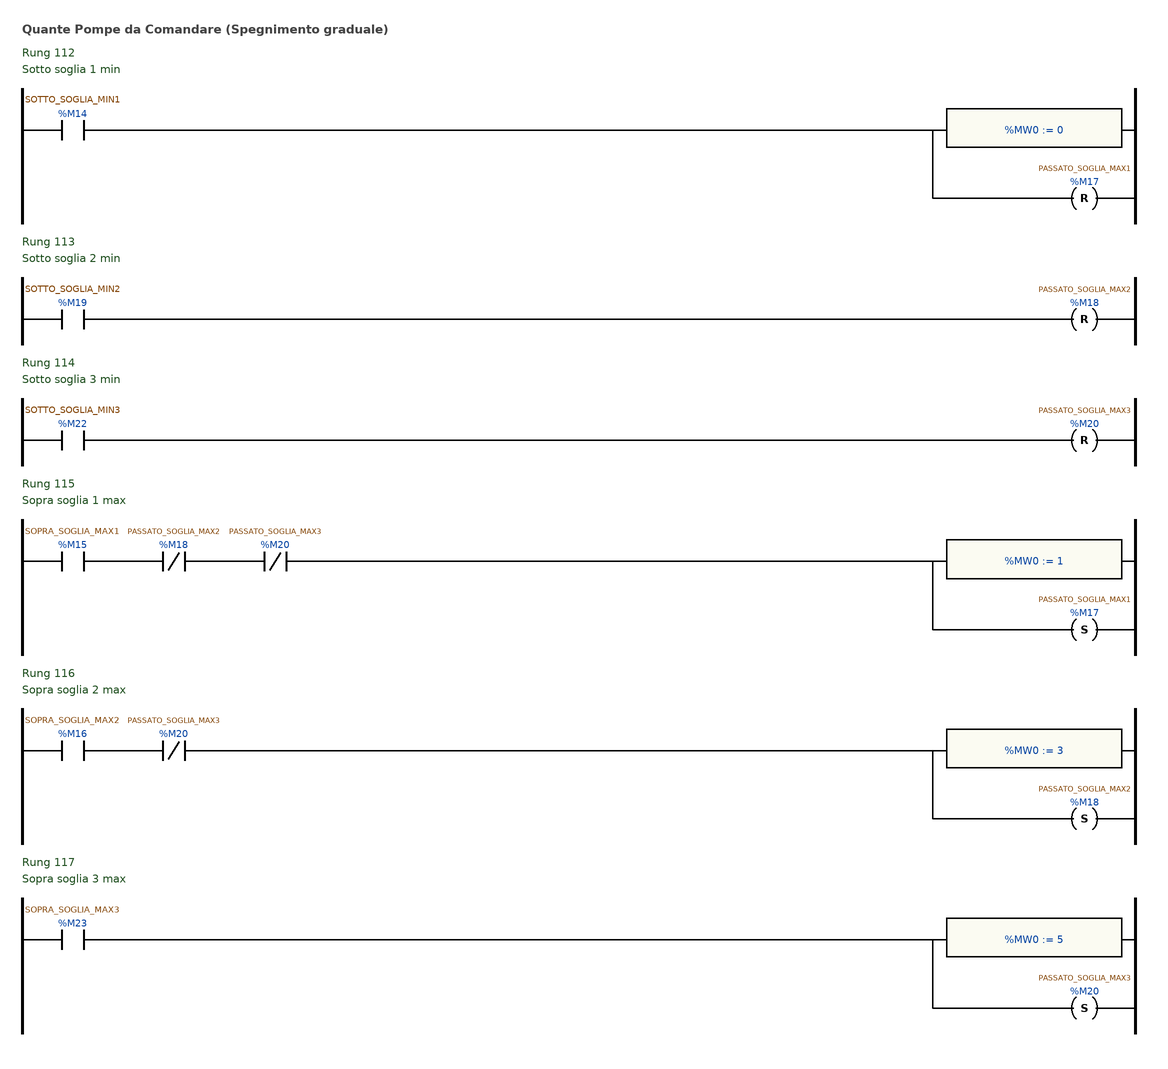
[picture p24: Quante Pompe da Comandare (Spegnimento graduale), ladder]

// Rung 112
// Sotto soglia 1 min
  LD %M14                 (* SOTTO_SOGLIA_MIN1 *)
  [ %MW0 := 0 ]           (* NUM_POMPE_DA_COMANDARE *)
  R %M17                  (* PASSATO_SOGLIA_MAX1 *)
  // as ST:
  //   IF SOTTO_SOGLIA_MIN1 THEN NUM_POMPE_DA_COMANDARE := 0; END_IF;
  //   IF SOTTO_SOGLIA_MIN1 THEN PASSATO_SOGLIA_MAX1 := FALSE; END_IF;

// Rung 113
// Sotto soglia 2 min
  LD %M19                 (* SOTTO_SOGLIA_MIN2 *)
  R %M18                  (* PASSATO_SOGLIA_MAX2 *)
  // as ST:
  //   IF SOTTO_SOGLIA_MIN2 THEN PASSATO_SOGLIA_MAX2 := FALSE; END_IF;

// Rung 114
// Sotto soglia 3 min
  LD %M22                 (* SOTTO_SOGLIA_MIN3 *)
  R %M20                  (* PASSATO_SOGLIA_MAX3 *)
  // as ST:
  //   IF SOTTO_SOGLIA_MIN3 THEN PASSATO_SOGLIA_MAX3 := FALSE; END_IF;

// Rung 115
// Sopra soglia 1 max
  LD %M15                 (* SOPRA_SOGLIA_MAX1 *)
  ANDN %M18               (* PASSATO_SOGLIA_MAX2 *)
  ANDN %M20               (* PASSATO_SOGLIA_MAX3 *)
  [ %MW0 := 1 ]           (* NUM_POMPE_DA_COMANDARE *)
  S %M17                  (* PASSATO_SOGLIA_MAX1 *)
  // as ST:
  //   IF SOPRA_SOGLIA_MAX1 AND NOT PASSATO_SOGLIA_MAX2 AND NOT PASSATO_SOGLIA_MAX3 THEN NUM_POMPE_DA_COMANDARE := 1; END_IF;
  //   IF SOPRA_SOGLIA_MAX1 AND NOT PASSATO_SOGLIA_MAX2 AND NOT PASSATO_SOGLIA_MAX3 THEN PASSATO_SOGLIA_MAX1 := TRUE; END_IF;

// Rung 116
// Sopra soglia 2 max
  LD %M16                 (* SOPRA_SOGLIA_MAX2 *)
  ANDN %M20               (* PASSATO_SOGLIA_MAX3 *)
  [ %MW0 := 3 ]           (* NUM_POMPE_DA_COMANDARE *)
  S %M18                  (* PASSATO_SOGLIA_MAX2 *)
  // as ST:
  //   IF SOPRA_SOGLIA_MAX2 AND NOT PASSATO_SOGLIA_MAX3 THEN NUM_POMPE_DA_COMANDARE := 3; END_IF;
  //   IF SOPRA_SOGLIA_MAX2 AND NOT PASSATO_SOGLIA_MAX3 THEN PASSATO_SOGLIA_MAX2 := TRUE; END_IF;

// Rung 117
// Sopra soglia 3 max
  LD %M23                 (* SOPRA_SOGLIA_MAX3 *)
  [ %MW0 := 5 ]           (* NUM_POMPE_DA_COMANDARE *)
  S %M20                  (* PASSATO_SOGLIA_MAX3 *)
  // as ST:
  //   IF SOPRA_SOGLIA_MAX3 THEN NUM_POMPE_DA_COMANDARE := 5; END_IF;
  //   IF SOPRA_SOGLIA_MAX3 THEN PASSATO_SOGLIA_MAX3 := TRUE; END_IF;

Subroutine Ordine: Quarta Pompa
  (* SectionNumber=16, Number=11 *)

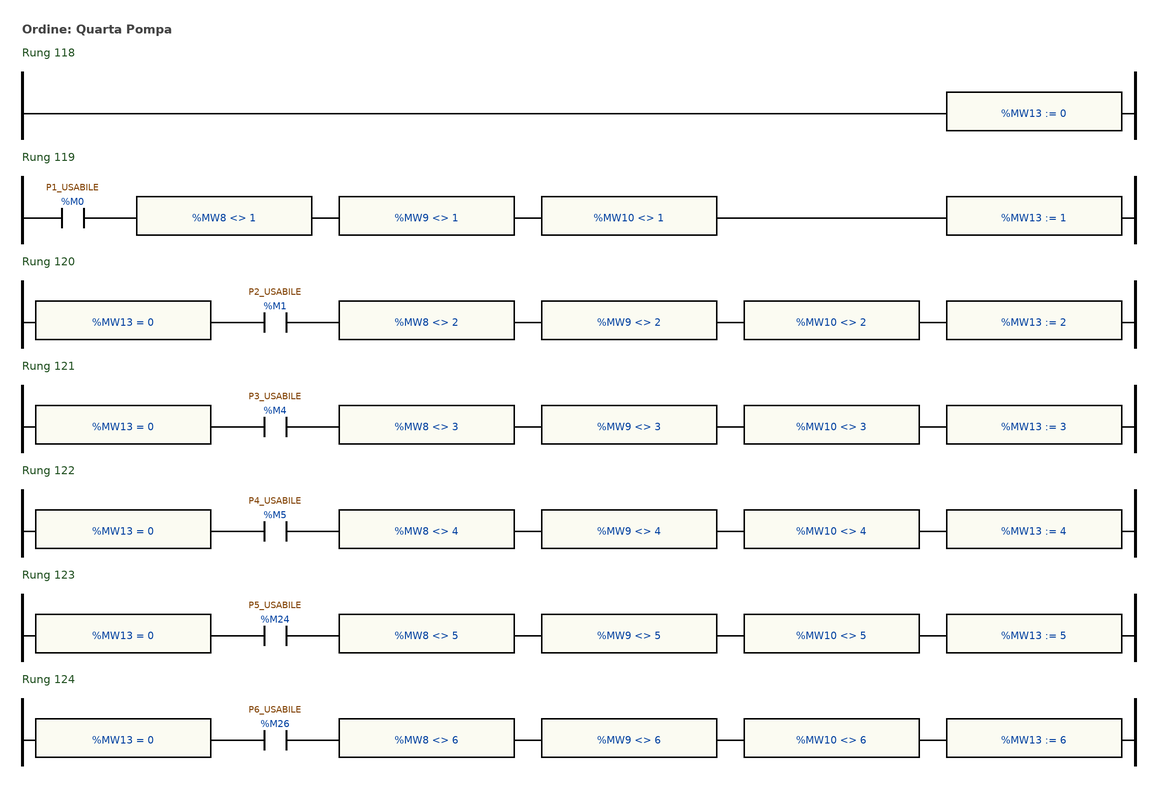

// Rung 118
  LD 1
  [ %MW13 := 0 ]          (* ORDINE_QUARTA_POMPA *)
  // as ST:
  //   ORDINE_QUARTA_POMPA := 0;

// Rung 119
  LD %M0                  (* P1_USABILE *)
  AND [ %MW8 <> 1 ]       (* ORDINE_PRIMA_POMPA *)
  AND [ %MW9 <> 1 ]       (* ORDINE_SECONDA_POMPA *)
  AND [ %MW10 <> 1 ]      (* ORDINE_TERZA_POMPA *)
  [ %MW13 := 1 ]          (* ORDINE_QUARTA_POMPA *)
  // as ST:
  //   IF P1_USABILE AND ORDINE_PRIMA_POMPA <> 1 AND ORDINE_SECONDA_POMPA <> 1 AND ORDINE_TERZA_POMPA <> 1 THEN ORDINE_QUARTA_POMPA := 1; END_IF;

// Rung 120
  LD [ %MW13 = 0 ]        (* ORDINE_QUARTA_POMPA *)
  AND %M1                 (* P2_USABILE *)
  AND [ %MW8 <> 2 ]       (* ORDINE_PRIMA_POMPA *)
  AND [ %MW9 <> 2 ]       (* ORDINE_SECONDA_POMPA *)
  AND [ %MW10 <> 2 ]      (* ORDINE_TERZA_POMPA *)
  [ %MW13 := 2 ]          (* ORDINE_QUARTA_POMPA *)
  // as ST:
  //   IF ORDINE_QUARTA_POMPA = 0 AND P2_USABILE AND ORDINE_PRIMA_POMPA <> 2 AND ORDINE_SECONDA_POMPA <> 2 AND ORDINE_TERZA_POMPA <> 2 THEN ORDINE_QUARTA_POMPA := 2; END_IF;

// Rung 121
  LD [ %MW13 = 0 ]        (* ORDINE_QUARTA_POMPA *)
  AND %M4                 (* P3_USABILE *)
  AND [ %MW8 <> 3 ]       (* ORDINE_PRIMA_POMPA *)
  AND [ %MW9 <> 3 ]       (* ORDINE_SECONDA_POMPA *)
  AND [ %MW10 <> 3 ]      (* ORDINE_TERZA_POMPA *)
  [ %MW13 := 3 ]          (* ORDINE_QUARTA_POMPA *)
  // as ST:
  //   IF ORDINE_QUARTA_POMPA = 0 AND P3_USABILE AND ORDINE_PRIMA_POMPA <> 3 AND ORDINE_SECONDA_POMPA <> 3 AND ORDINE_TERZA_POMPA <> 3 THEN ORDINE_QUARTA_POMPA := 3; END_IF;

// Rung 122
  LD [ %MW13 = 0 ]        (* ORDINE_QUARTA_POMPA *)
  AND %M5                 (* P4_USABILE *)
  AND [ %MW8 <> 4 ]       (* ORDINE_PRIMA_POMPA *)
  AND [ %MW9 <> 4 ]       (* ORDINE_SECONDA_POMPA *)
  AND [ %MW10 <> 4 ]      (* ORDINE_TERZA_POMPA *)
  [ %MW13 := 4 ]          (* ORDINE_QUARTA_POMPA *)
  // as ST:
  //   IF ORDINE_QUARTA_POMPA = 0 AND P4_USABILE AND ORDINE_PRIMA_POMPA <> 4 AND ORDINE_SECONDA_POMPA <> 4 AND ORDINE_TERZA_POMPA <> 4 THEN ORDINE_QUARTA_POMPA := 4; END_IF;

// Rung 123
  LD [ %MW13 = 0 ]        (* ORDINE_QUARTA_POMPA *)
  AND %M24                (* P5_USABILE *)
  AND [ %MW8 <> 5 ]       (* ORDINE_PRIMA_POMPA *)
  AND [ %MW9 <> 5 ]       (* ORDINE_SECONDA_POMPA *)
  AND [ %MW10 <> 5 ]      (* ORDINE_TERZA_POMPA *)
  [ %MW13 := 5 ]          (* ORDINE_QUARTA_POMPA *)
  // as ST:
  //   IF ORDINE_QUARTA_POMPA = 0 AND P5_USABILE AND ORDINE_PRIMA_POMPA <> 5 AND ORDINE_SECONDA_POMPA <> 5 AND ORDINE_TERZA_POMPA <> 5 THEN ORDINE_QUARTA_POMPA := 5; END_IF;

// Rung 124
  LD [ %MW13 = 0 ]        (* ORDINE_QUARTA_POMPA *)
  AND %M26                (* P6_USABILE *)
  AND [ %MW8 <> 6 ]       (* ORDINE_PRIMA_POMPA *)
  AND [ %MW9 <> 6 ]       (* ORDINE_SECONDA_POMPA *)
  AND [ %MW10 <> 6 ]      (* ORDINE_TERZA_POMPA *)
  [ %MW13 := 6 ]          (* ORDINE_QUARTA_POMPA *)
  // as ST:
  //   IF ORDINE_QUARTA_POMPA = 0 AND P6_USABILE AND ORDINE_PRIMA_POMPA <> 6 AND ORDINE_SECONDA_POMPA <> 6 AND ORDINE_TERZA_POMPA <> 6 THEN ORDINE_QUARTA_POMPA := 6; END_IF;

Subroutine Ordine: Quinta Pompa
  (* SectionNumber=17, Number=12 *)

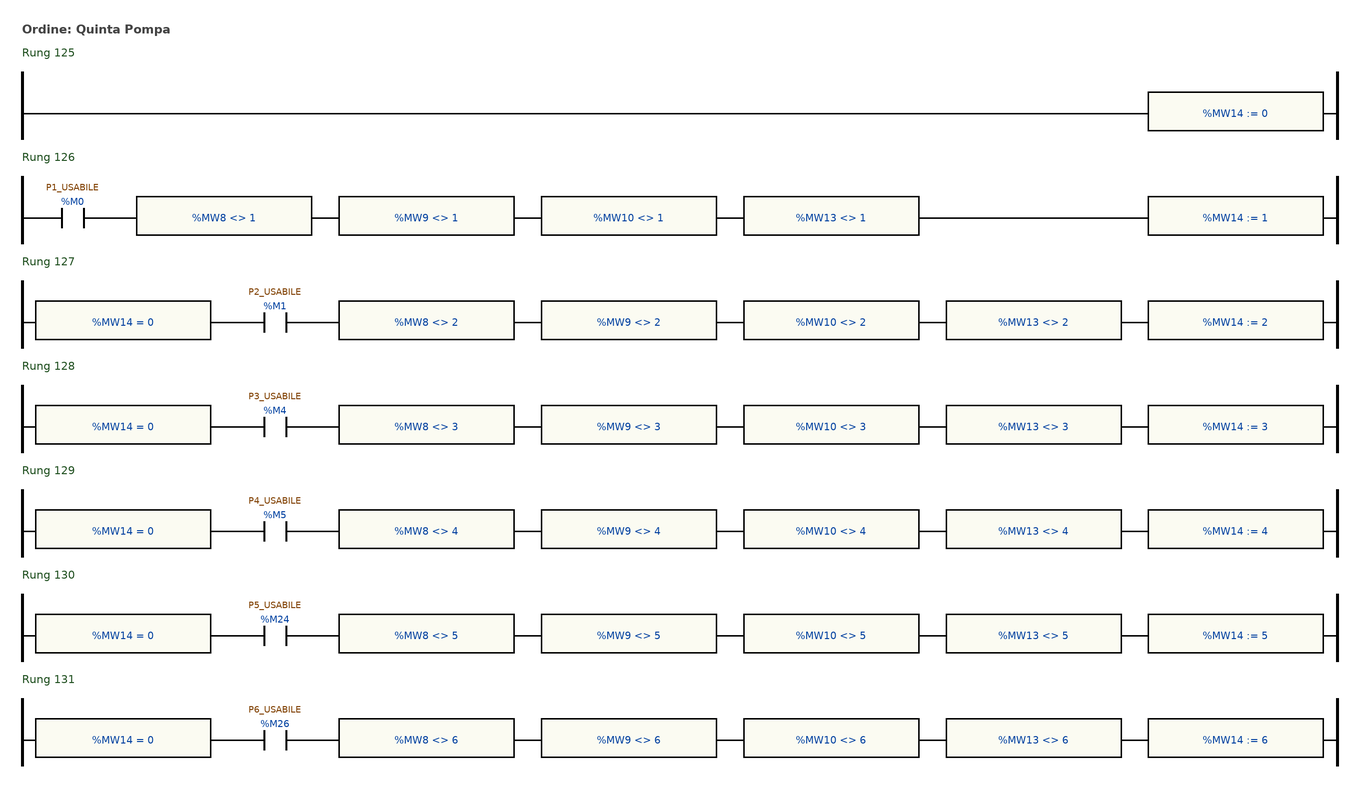

// Rung 125
  LD 1
  [ %MW14 := 0 ]          (* ORDINE_QUINTA_POMPA *)
  // as ST:
  //   ORDINE_QUINTA_POMPA := 0;

// Rung 126
  LD %M0                  (* P1_USABILE *)
  AND [ %MW8 <> 1 ]       (* ORDINE_PRIMA_POMPA *)
  AND [ %MW9 <> 1 ]       (* ORDINE_SECONDA_POMPA *)
  AND [ %MW10 <> 1 ]      (* ORDINE_TERZA_POMPA *)
  AND [ %MW13 <> 1 ]      (* ORDINE_QUARTA_POMPA *)
  [ %MW14 := 1 ]          (* ORDINE_QUINTA_POMPA *)
  // as ST:
  //   IF P1_USABILE AND ORDINE_PRIMA_POMPA <> 1 AND ORDINE_SECONDA_POMPA <> 1 AND ORDINE_TERZA_POMPA <> 1 AND ORDINE_QUARTA_POMPA <> 1 THEN ORDINE_QUINTA_POMPA := 1; END_IF;

// Rung 127
  LD [ %MW14 = 0 ]        (* ORDINE_QUINTA_POMPA *)
  AND %M1                 (* P2_USABILE *)
  AND [ %MW8 <> 2 ]       (* ORDINE_PRIMA_POMPA *)
  AND [ %MW9 <> 2 ]       (* ORDINE_SECONDA_POMPA *)
  AND [ %MW10 <> 2 ]      (* ORDINE_TERZA_POMPA *)
  AND [ %MW13 <> 2 ]      (* ORDINE_QUARTA_POMPA *)
  [ %MW14 := 2 ]          (* ORDINE_QUINTA_POMPA *)
  // as ST:
  //   IF ORDINE_QUINTA_POMPA = 0 AND P2_USABILE AND ORDINE_PRIMA_POMPA <> 2 AND ORDINE_SECONDA_POMPA <> 2 AND ORDINE_TERZA_POMPA <> 2 AND ORDINE_QUARTA_POMPA <> 2 THEN ORDINE_QUINTA_POMPA := 2; END_IF;

// Rung 128
  LD [ %MW14 = 0 ]        (* ORDINE_QUINTA_POMPA *)
  AND %M4                 (* P3_USABILE *)
  AND [ %MW8 <> 3 ]       (* ORDINE_PRIMA_POMPA *)
  AND [ %MW9 <> 3 ]       (* ORDINE_SECONDA_POMPA *)
  AND [ %MW10 <> 3 ]      (* ORDINE_TERZA_POMPA *)
  AND [ %MW13 <> 3 ]      (* ORDINE_QUARTA_POMPA *)
  [ %MW14 := 3 ]          (* ORDINE_QUINTA_POMPA *)
  // as ST:
  //   IF ORDINE_QUINTA_POMPA = 0 AND P3_USABILE AND ORDINE_PRIMA_POMPA <> 3 AND ORDINE_SECONDA_POMPA <> 3 AND ORDINE_TERZA_POMPA <> 3 AND ORDINE_QUARTA_POMPA <> 3 THEN ORDINE_QUINTA_POMPA := 3; END_IF;

// Rung 129
  LD [ %MW14 = 0 ]        (* ORDINE_QUINTA_POMPA *)
  AND %M5                 (* P4_USABILE *)
  AND [ %MW8 <> 4 ]       (* ORDINE_PRIMA_POMPA *)
  AND [ %MW9 <> 4 ]       (* ORDINE_SECONDA_POMPA *)
  AND [ %MW10 <> 4 ]      (* ORDINE_TERZA_POMPA *)
  AND [ %MW13 <> 4 ]      (* ORDINE_QUARTA_POMPA *)
  [ %MW14 := 4 ]          (* ORDINE_QUINTA_POMPA *)
  // as ST:
  //   IF ORDINE_QUINTA_POMPA = 0 AND P4_USABILE AND ORDINE_PRIMA_POMPA <> 4 AND ORDINE_SECONDA_POMPA <> 4 AND ORDINE_TERZA_POMPA <> 4 AND ORDINE_QUARTA_POMPA <> 4 THEN ORDINE_QUINTA_POMPA := 4; END_IF;

// Rung 130
  LD [ %MW14 = 0 ]        (* ORDINE_QUINTA_POMPA *)
  AND %M24                (* P5_USABILE *)
  AND [ %MW8 <> 5 ]       (* ORDINE_PRIMA_POMPA *)
  AND [ %MW9 <> 5 ]       (* ORDINE_SECONDA_POMPA *)
  AND [ %MW10 <> 5 ]      (* ORDINE_TERZA_POMPA *)
  AND [ %MW13 <> 5 ]      (* ORDINE_QUARTA_POMPA *)
  [ %MW14 := 5 ]          (* ORDINE_QUINTA_POMPA *)
  // as ST:
  //   IF ORDINE_QUINTA_POMPA = 0 AND P5_USABILE AND ORDINE_PRIMA_POMPA <> 5 AND ORDINE_SECONDA_POMPA <> 5 AND ORDINE_TERZA_POMPA <> 5 AND ORDINE_QUARTA_POMPA <> 5 THEN ORDINE_QUINTA_POMPA := 5; END_IF;

// Rung 131
  LD [ %MW14 = 0 ]        (* ORDINE_QUINTA_POMPA *)
  AND %M26                (* P6_USABILE *)
  AND [ %MW8 <> 6 ]       (* ORDINE_PRIMA_POMPA *)
  AND [ %MW9 <> 6 ]       (* ORDINE_SECONDA_POMPA *)
  AND [ %MW10 <> 6 ]      (* ORDINE_TERZA_POMPA *)
  AND [ %MW13 <> 6 ]      (* ORDINE_QUARTA_POMPA *)
  [ %MW14 := 6 ]          (* ORDINE_QUINTA_POMPA *)
  // as ST:
  //   IF ORDINE_QUINTA_POMPA = 0 AND P6_USABILE AND ORDINE_PRIMA_POMPA <> 6 AND ORDINE_SECONDA_POMPA <> 6 AND ORDINE_TERZA_POMPA <> 6 AND ORDINE_QUARTA_POMPA <> 6 THEN ORDINE_QUINTA_POMPA := 6; END_IF;

Subroutine Comanda: Quarta Pompa
  (* SectionNumber=18, Number=14 *)

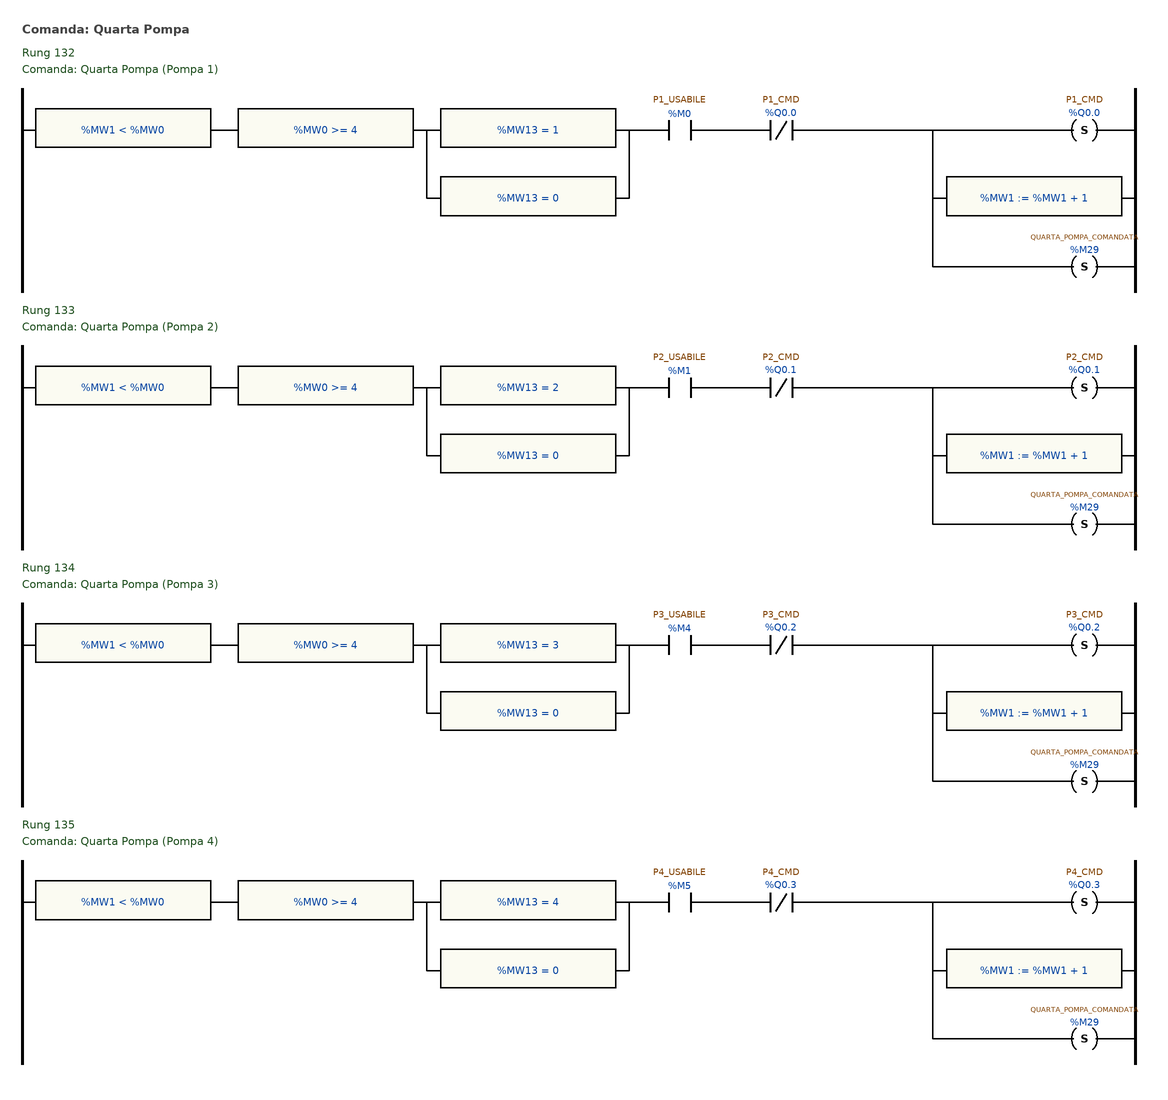

// Rung 132
// Comanda: Quarta Pompa (Pompa 1)
  LD [ %MW1 < %MW0 ]      (* NUM_POMPE_COMANDATE, NUM_POMPE_DA_COMANDARE *)
  AND [ %MW0 >= 4 ]       (* NUM_POMPE_DA_COMANDARE *)
  AND( [ %MW13 = 1 ]      (* ORDINE_QUARTA_POMPA *)
  OR [ %MW13 = 0 ]        (* ORDINE_QUARTA_POMPA *)
  )
  AND %M0                 (* P1_USABILE *)
  ANDN %Q0.0              (* P1_CMD *)
  S %Q0.0                 (* P1_CMD *)
  [ %MW1 := %MW1 + 1 ]    (* NUM_POMPE_COMANDATE, NUM_POMPE_COMANDATE *)
  S %M29                  (* QUARTA_POMPA_COMANDATA *)
  // as ST:
  //   _t1 := NUM_POMPE_COMANDATE < NUM_POMPE_DA_COMANDARE AND NUM_POMPE_DA_COMANDARE >= 4 AND (ORDINE_QUARTA_POMPA = 1 OR ORDINE_QUARTA_POMPA = 0) AND P1_USABILE AND NOT P1_CMD;
  //   IF _t1 THEN P1_CMD := TRUE; END_IF;
  //   IF _t1 THEN NUM_POMPE_COMANDATE := NUM_POMPE_COMANDATE + 1; END_IF;
  //   IF _t1 THEN QUARTA_POMPA_COMANDATA := TRUE; END_IF;

// Rung 133
// Comanda: Quarta Pompa (Pompa 2)
  LD [ %MW1 < %MW0 ]      (* NUM_POMPE_COMANDATE, NUM_POMPE_DA_COMANDARE *)
  AND [ %MW0 >= 4 ]       (* NUM_POMPE_DA_COMANDARE *)
  AND( [ %MW13 = 2 ]      (* ORDINE_QUARTA_POMPA *)
  OR [ %MW13 = 0 ]        (* ORDINE_QUARTA_POMPA *)
  )
  AND %M1                 (* P2_USABILE *)
  ANDN %Q0.1              (* P2_CMD *)
  S %Q0.1                 (* P2_CMD *)
  [ %MW1 := %MW1 + 1 ]    (* NUM_POMPE_COMANDATE, NUM_POMPE_COMANDATE *)
  S %M29                  (* QUARTA_POMPA_COMANDATA *)
  // as ST:
  //   _t1 := NUM_POMPE_COMANDATE < NUM_POMPE_DA_COMANDARE AND NUM_POMPE_DA_COMANDARE >= 4 AND (ORDINE_QUARTA_POMPA = 2 OR ORDINE_QUARTA_POMPA = 0) AND P2_USABILE AND NOT P2_CMD;
  //   IF _t1 THEN P2_CMD := TRUE; END_IF;
  //   IF _t1 THEN NUM_POMPE_COMANDATE := NUM_POMPE_COMANDATE + 1; END_IF;
  //   IF _t1 THEN QUARTA_POMPA_COMANDATA := TRUE; END_IF;

// Rung 134
// Comanda: Quarta Pompa (Pompa 3)
  LD [ %MW1 < %MW0 ]      (* NUM_POMPE_COMANDATE, NUM_POMPE_DA_COMANDARE *)
  AND [ %MW0 >= 4 ]       (* NUM_POMPE_DA_COMANDARE *)
  AND( [ %MW13 = 3 ]      (* ORDINE_QUARTA_POMPA *)
  OR [ %MW13 = 0 ]        (* ORDINE_QUARTA_POMPA *)
  )
  AND %M4                 (* P3_USABILE *)
  ANDN %Q0.2              (* P3_CMD *)
  S %Q0.2                 (* P3_CMD *)
  [ %MW1 := %MW1 + 1 ]    (* NUM_POMPE_COMANDATE, NUM_POMPE_COMANDATE *)
  S %M29                  (* QUARTA_POMPA_COMANDATA *)
  // as ST:
  //   _t1 := NUM_POMPE_COMANDATE < NUM_POMPE_DA_COMANDARE AND NUM_POMPE_DA_COMANDARE >= 4 AND (ORDINE_QUARTA_POMPA = 3 OR ORDINE_QUARTA_POMPA = 0) AND P3_USABILE AND NOT P3_CMD;
  //   IF _t1 THEN P3_CMD := TRUE; END_IF;
  //   IF _t1 THEN NUM_POMPE_COMANDATE := NUM_POMPE_COMANDATE + 1; END_IF;
  //   IF _t1 THEN QUARTA_POMPA_COMANDATA := TRUE; END_IF;

// Rung 135
// Comanda: Quarta Pompa (Pompa 4)
  LD [ %MW1 < %MW0 ]      (* NUM_POMPE_COMANDATE, NUM_POMPE_DA_COMANDARE *)
  AND [ %MW0 >= 4 ]       (* NUM_POMPE_DA_COMANDARE *)
  AND( [ %MW13 = 4 ]      (* ORDINE_QUARTA_POMPA *)
  OR [ %MW13 = 0 ]        (* ORDINE_QUARTA_POMPA *)
  )
  AND %M5                 (* P4_USABILE *)
  ANDN %Q0.3              (* P4_CMD *)
  S %Q0.3                 (* P4_CMD *)
  [ %MW1 := %MW1 + 1 ]    (* NUM_POMPE_COMANDATE, NUM_POMPE_COMANDATE *)
  S %M29                  (* QUARTA_POMPA_COMANDATA *)
  // as ST:
  //   _t1 := NUM_POMPE_COMANDATE < NUM_POMPE_DA_COMANDARE AND NUM_POMPE_DA_COMANDARE >= 4 AND (ORDINE_QUARTA_POMPA = 4 OR ORDINE_QUARTA_POMPA = 0) AND P4_USABILE AND NOT P4_CMD;
  //   IF _t1 THEN P4_CMD := TRUE; END_IF;
  //   IF _t1 THEN NUM_POMPE_COMANDATE := NUM_POMPE_COMANDATE + 1; END_IF;
  //   IF _t1 THEN QUARTA_POMPA_COMANDATA := TRUE; END_IF;

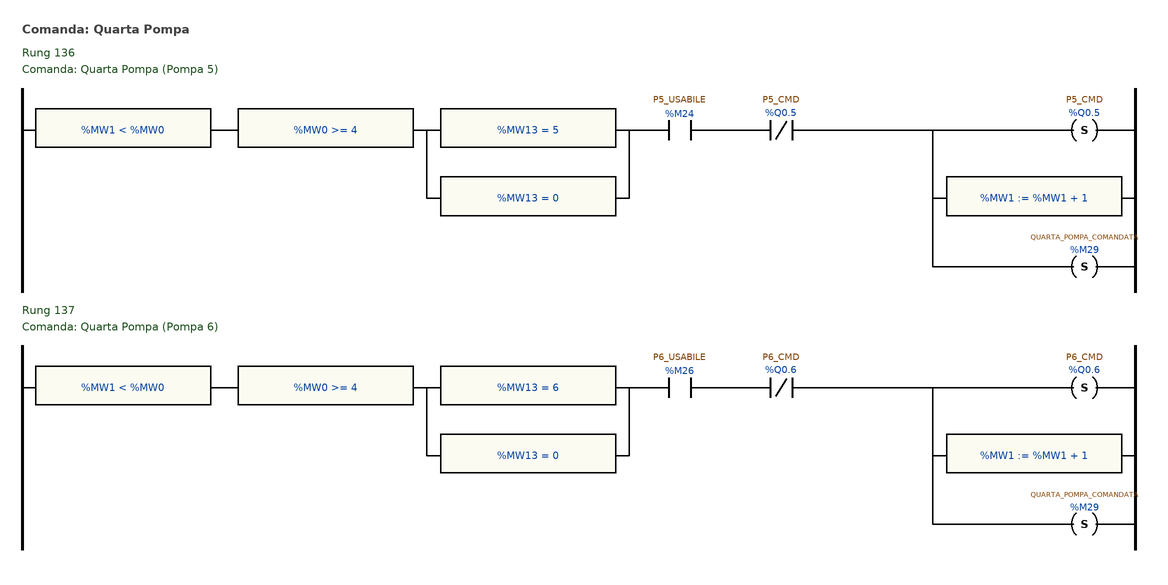

// Rung 136
// Comanda: Quarta Pompa (Pompa 5)
  LD [ %MW1 < %MW0 ]      (* NUM_POMPE_COMANDATE, NUM_POMPE_DA_COMANDARE *)
  AND [ %MW0 >= 4 ]       (* NUM_POMPE_DA_COMANDARE *)
  AND( [ %MW13 = 5 ]      (* ORDINE_QUARTA_POMPA *)
  OR [ %MW13 = 0 ]        (* ORDINE_QUARTA_POMPA *)
  )
  AND %M24                (* P5_USABILE *)
  ANDN %Q0.5              (* P5_CMD *)
  S %Q0.5                 (* P5_CMD *)
  [ %MW1 := %MW1 + 1 ]    (* NUM_POMPE_COMANDATE, NUM_POMPE_COMANDATE *)
  S %M29                  (* QUARTA_POMPA_COMANDATA *)
  // as ST:
  //   _t1 := NUM_POMPE_COMANDATE < NUM_POMPE_DA_COMANDARE AND NUM_POMPE_DA_COMANDARE >= 4 AND (ORDINE_QUARTA_POMPA = 5 OR ORDINE_QUARTA_POMPA = 0) AND P5_USABILE AND NOT P5_CMD;
  //   IF _t1 THEN P5_CMD := TRUE; END_IF;
  //   IF _t1 THEN NUM_POMPE_COMANDATE := NUM_POMPE_COMANDATE + 1; END_IF;
  //   IF _t1 THEN QUARTA_POMPA_COMANDATA := TRUE; END_IF;

// Rung 137
// Comanda: Quarta Pompa (Pompa 6)
  LD [ %MW1 < %MW0 ]      (* NUM_POMPE_COMANDATE, NUM_POMPE_DA_COMANDARE *)
  AND [ %MW0 >= 4 ]       (* NUM_POMPE_DA_COMANDARE *)
  AND( [ %MW13 = 6 ]      (* ORDINE_QUARTA_POMPA *)
  OR [ %MW13 = 0 ]        (* ORDINE_QUARTA_POMPA *)
  )
  AND %M26                (* P6_USABILE *)
  ANDN %Q0.6              (* P6_CMD *)
  S %Q0.6                 (* P6_CMD *)
  [ %MW1 := %MW1 + 1 ]    (* NUM_POMPE_COMANDATE, NUM_POMPE_COMANDATE *)
  S %M29                  (* QUARTA_POMPA_COMANDATA *)
  // as ST:
  //   _t1 := NUM_POMPE_COMANDATE < NUM_POMPE_DA_COMANDARE AND NUM_POMPE_DA_COMANDARE >= 4 AND (ORDINE_QUARTA_POMPA = 6 OR ORDINE_QUARTA_POMPA = 0) AND P6_USABILE AND NOT P6_CMD;
  //   IF _t1 THEN P6_CMD := TRUE; END_IF;
  //   IF _t1 THEN NUM_POMPE_COMANDATE := NUM_POMPE_COMANDATE + 1; END_IF;
  //   IF _t1 THEN QUARTA_POMPA_COMANDATA := TRUE; END_IF;

Subroutine Comanda: Quinta Pompa
  (* SectionNumber=19, Number=15 *)

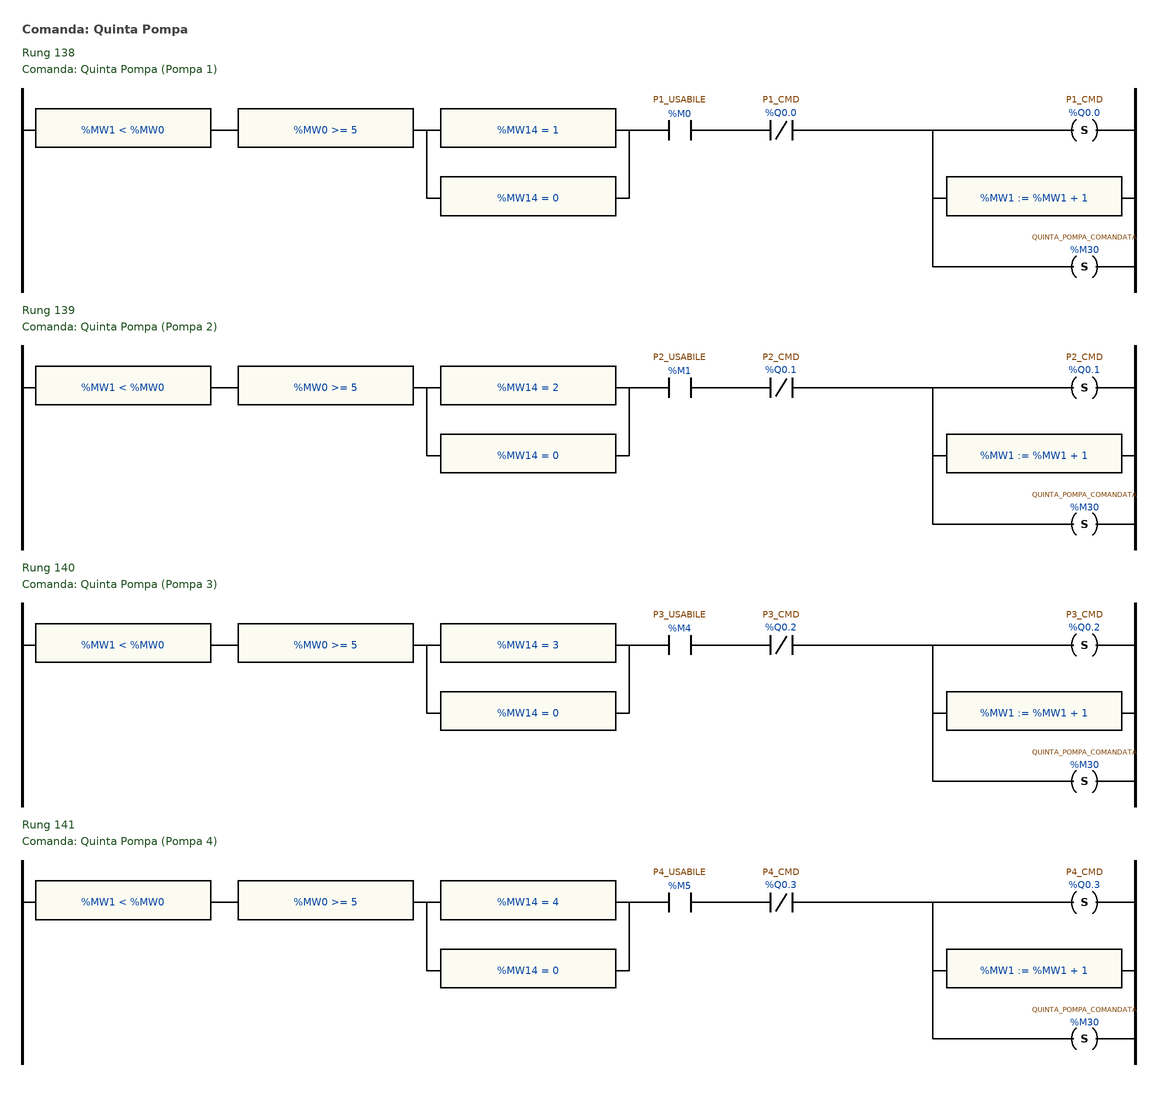

// Rung 138
// Comanda: Quinta Pompa (Pompa 1)
  LD [ %MW1 < %MW0 ]      (* NUM_POMPE_COMANDATE, NUM_POMPE_DA_COMANDARE *)
  AND [ %MW0 >= 5 ]       (* NUM_POMPE_DA_COMANDARE *)
  AND( [ %MW14 = 1 ]      (* ORDINE_QUINTA_POMPA *)
  OR [ %MW14 = 0 ]        (* ORDINE_QUINTA_POMPA *)
  )
  AND %M0                 (* P1_USABILE *)
  ANDN %Q0.0              (* P1_CMD *)
  S %Q0.0                 (* P1_CMD *)
  [ %MW1 := %MW1 + 1 ]    (* NUM_POMPE_COMANDATE, NUM_POMPE_COMANDATE *)
  S %M30                  (* QUINTA_POMPA_COMANDATA *)
  // as ST:
  //   _t1 := NUM_POMPE_COMANDATE < NUM_POMPE_DA_COMANDARE AND NUM_POMPE_DA_COMANDARE >= 5 AND (ORDINE_QUINTA_POMPA = 1 OR ORDINE_QUINTA_POMPA = 0) AND P1_USABILE AND NOT P1_CMD;
  //   IF _t1 THEN P1_CMD := TRUE; END_IF;
  //   IF _t1 THEN NUM_POMPE_COMANDATE := NUM_POMPE_COMANDATE + 1; END_IF;
  //   IF _t1 THEN QUINTA_POMPA_COMANDATA := TRUE; END_IF;

// Rung 139
// Comanda: Quinta Pompa (Pompa 2)
  LD [ %MW1 < %MW0 ]      (* NUM_POMPE_COMANDATE, NUM_POMPE_DA_COMANDARE *)
  AND [ %MW0 >= 5 ]       (* NUM_POMPE_DA_COMANDARE *)
  AND( [ %MW14 = 2 ]      (* ORDINE_QUINTA_POMPA *)
  OR [ %MW14 = 0 ]        (* ORDINE_QUINTA_POMPA *)
  )
  AND %M1                 (* P2_USABILE *)
  ANDN %Q0.1              (* P2_CMD *)
  S %Q0.1                 (* P2_CMD *)
  [ %MW1 := %MW1 + 1 ]    (* NUM_POMPE_COMANDATE, NUM_POMPE_COMANDATE *)
  S %M30                  (* QUINTA_POMPA_COMANDATA *)
  // as ST:
  //   _t1 := NUM_POMPE_COMANDATE < NUM_POMPE_DA_COMANDARE AND NUM_POMPE_DA_COMANDARE >= 5 AND (ORDINE_QUINTA_POMPA = 2 OR ORDINE_QUINTA_POMPA = 0) AND P2_USABILE AND NOT P2_CMD;
  //   IF _t1 THEN P2_CMD := TRUE; END_IF;
  //   IF _t1 THEN NUM_POMPE_COMANDATE := NUM_POMPE_COMANDATE + 1; END_IF;
  //   IF _t1 THEN QUINTA_POMPA_COMANDATA := TRUE; END_IF;

// Rung 140
// Comanda: Quinta Pompa (Pompa 3)
  LD [ %MW1 < %MW0 ]      (* NUM_POMPE_COMANDATE, NUM_POMPE_DA_COMANDARE *)
  AND [ %MW0 >= 5 ]       (* NUM_POMPE_DA_COMANDARE *)
  AND( [ %MW14 = 3 ]      (* ORDINE_QUINTA_POMPA *)
  OR [ %MW14 = 0 ]        (* ORDINE_QUINTA_POMPA *)
  )
  AND %M4                 (* P3_USABILE *)
  ANDN %Q0.2              (* P3_CMD *)
  S %Q0.2                 (* P3_CMD *)
  [ %MW1 := %MW1 + 1 ]    (* NUM_POMPE_COMANDATE, NUM_POMPE_COMANDATE *)
  S %M30                  (* QUINTA_POMPA_COMANDATA *)
  // as ST:
  //   _t1 := NUM_POMPE_COMANDATE < NUM_POMPE_DA_COMANDARE AND NUM_POMPE_DA_COMANDARE >= 5 AND (ORDINE_QUINTA_POMPA = 3 OR ORDINE_QUINTA_POMPA = 0) AND P3_USABILE AND NOT P3_CMD;
  //   IF _t1 THEN P3_CMD := TRUE; END_IF;
  //   IF _t1 THEN NUM_POMPE_COMANDATE := NUM_POMPE_COMANDATE + 1; END_IF;
  //   IF _t1 THEN QUINTA_POMPA_COMANDATA := TRUE; END_IF;

// Rung 141
// Comanda: Quinta Pompa (Pompa 4)
  LD [ %MW1 < %MW0 ]      (* NUM_POMPE_COMANDATE, NUM_POMPE_DA_COMANDARE *)
  AND [ %MW0 >= 5 ]       (* NUM_POMPE_DA_COMANDARE *)
  AND( [ %MW14 = 4 ]      (* ORDINE_QUINTA_POMPA *)
  OR [ %MW14 = 0 ]        (* ORDINE_QUINTA_POMPA *)
  )
  AND %M5                 (* P4_USABILE *)
  ANDN %Q0.3              (* P4_CMD *)
  S %Q0.3                 (* P4_CMD *)
  [ %MW1 := %MW1 + 1 ]    (* NUM_POMPE_COMANDATE, NUM_POMPE_COMANDATE *)
  S %M30                  (* QUINTA_POMPA_COMANDATA *)
  // as ST:
  //   _t1 := NUM_POMPE_COMANDATE < NUM_POMPE_DA_COMANDARE AND NUM_POMPE_DA_COMANDARE >= 5 AND (ORDINE_QUINTA_POMPA = 4 OR ORDINE_QUINTA_POMPA = 0) AND P4_USABILE AND NOT P4_CMD;
  //   IF _t1 THEN P4_CMD := TRUE; END_IF;
  //   IF _t1 THEN NUM_POMPE_COMANDATE := NUM_POMPE_COMANDATE + 1; END_IF;
  //   IF _t1 THEN QUINTA_POMPA_COMANDATA := TRUE; END_IF;

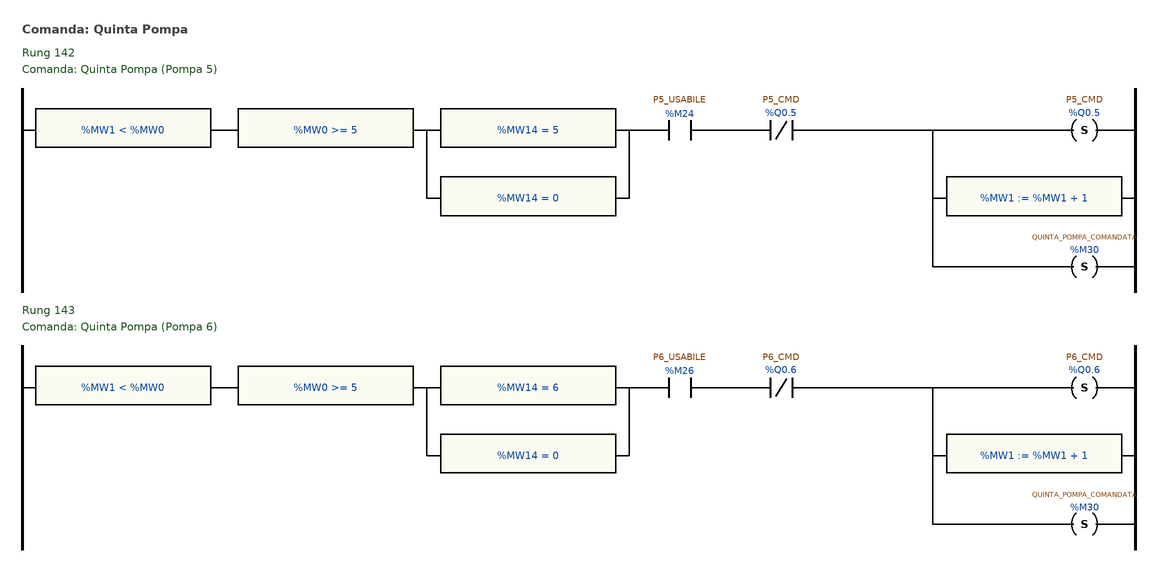

// Rung 142
// Comanda: Quinta Pompa (Pompa 5)
  LD [ %MW1 < %MW0 ]      (* NUM_POMPE_COMANDATE, NUM_POMPE_DA_COMANDARE *)
  AND [ %MW0 >= 5 ]       (* NUM_POMPE_DA_COMANDARE *)
  AND( [ %MW14 = 5 ]      (* ORDINE_QUINTA_POMPA *)
  OR [ %MW14 = 0 ]        (* ORDINE_QUINTA_POMPA *)
  )
  AND %M24                (* P5_USABILE *)
  ANDN %Q0.5              (* P5_CMD *)
  S %Q0.5                 (* P5_CMD *)
  [ %MW1 := %MW1 + 1 ]    (* NUM_POMPE_COMANDATE, NUM_POMPE_COMANDATE *)
  S %M30                  (* QUINTA_POMPA_COMANDATA *)
  // as ST:
  //   _t1 := NUM_POMPE_COMANDATE < NUM_POMPE_DA_COMANDARE AND NUM_POMPE_DA_COMANDARE >= 5 AND (ORDINE_QUINTA_POMPA = 5 OR ORDINE_QUINTA_POMPA = 0) AND P5_USABILE AND NOT P5_CMD;
  //   IF _t1 THEN P5_CMD := TRUE; END_IF;
  //   IF _t1 THEN NUM_POMPE_COMANDATE := NUM_POMPE_COMANDATE + 1; END_IF;
  //   IF _t1 THEN QUINTA_POMPA_COMANDATA := TRUE; END_IF;

// Rung 143
// Comanda: Quinta Pompa (Pompa 6)
  LD [ %MW1 < %MW0 ]      (* NUM_POMPE_COMANDATE, NUM_POMPE_DA_COMANDARE *)
  AND [ %MW0 >= 5 ]       (* NUM_POMPE_DA_COMANDARE *)
  AND( [ %MW14 = 6 ]      (* ORDINE_QUINTA_POMPA *)
  OR [ %MW14 = 0 ]        (* ORDINE_QUINTA_POMPA *)
  )
  AND %M26                (* P6_USABILE *)
  ANDN %Q0.6              (* P6_CMD *)
  S %Q0.6                 (* P6_CMD *)
  [ %MW1 := %MW1 + 1 ]    (* NUM_POMPE_COMANDATE, NUM_POMPE_COMANDATE *)
  S %M30                  (* QUINTA_POMPA_COMANDATA *)
  // as ST:
  //   _t1 := NUM_POMPE_COMANDATE < NUM_POMPE_DA_COMANDARE AND NUM_POMPE_DA_COMANDARE >= 5 AND (ORDINE_QUINTA_POMPA = 6 OR ORDINE_QUINTA_POMPA = 0) AND P6_USABILE AND NOT P6_CMD;
  //   IF _t1 THEN P6_CMD := TRUE; END_IF;
  //   IF _t1 THEN NUM_POMPE_COMANDATE := NUM_POMPE_COMANDATE + 1; END_IF;
  //   IF _t1 THEN QUINTA_POMPA_COMANDATA := TRUE; END_IF;
